INTERFACE I_PackML_Module

METHOD ChangeMode
VAR_INPUT
	RequestedMode : DINT;
END_VAR
END_METHOD

METHOD ChangeState
VAR_INPUT
	StateCommand : E_PMLCommand;
END_VAR
END_METHOD

{attribute 'monitoring' := 'call'}
PROPERTY CurrentMode : DINT
GET
END_GET
END_PROPERTY

{attribute 'monitoring' := 'call'}
PROPERTY CurrentState : E_PMLState
GET
END_GET
END_PROPERTY

{attribute 'monitoring' := 'call'}
PROPERTY Name : T_MaxString
GET
END_GET
SET
END_SET
END_PROPERTY

END_INTERFACE

(* stored: Version 1.1.0.1, ProductVersion 3.1.4026.18
   Itf I_PackML_Module: Id {7b001dc0-f9db-40cb-b066-2f920fd9874a}
   Method ChangeMode: Id {9f9a492c-3617-4d5c-9edf-64f53d46f8cb}
   Method ChangeState: Id {3913882f-b048-4a5b-93a4-23d3100b29b0}
   Property CurrentMode: Id {0165e033-657f-46c0-bb2c-2b22ba5c4c88}
   Get Get: Id {7345c78b-d44d-459c-a6ed-ac02999b293a}
   Property CurrentState: Id {b9d1fb52-23d7-4857-9742-d5e2e0b31192}
   Get Get: Id {e2bcd4f6-2a89-4d4b-93fa-7e9eee597592}
   Property Name: Id {848440c2-33f1-4786-a861-a09db7b9c76f}
   Get Get: Id {0ca88c35-2bea-41e1-b435-d95d16080f1e}
   Set Set: Id {3bef0a0c-a3ea-40f7-b1a6-62bed578d737} *)
